TEXTLIST LevelCmbTxtList
  1 = '1'
  2 = '2'
  3 = '3'
  4 = '4'
  5 = '5'
  6 = '6'
  7 = '7'
  8 = '8'
  9 = '9'
  10 = '10'
  11 = '11'
  12 = '12'
   = ''
END_TEXTLIST

(* stored: Version 1.1.0.1, ProductVersion 3.1.4024.4
   TextList LevelCmbTxtList: Id {1575c2e0-a107-4d2d-81b1-c1572076001f} *)
